PROGRAM P_Dialog
VAR
	nXPos 			: INT:=200; //pozycja popup na ekranie
	nYPos 			: INT:=200; //pozycja popup na ekranie
	fbOpenTrigger 	: R_TRIG;
	bClose 			: BOOL;
	fbCloseTrigger 	: R_TRIG;
	sMessage		: STRING;
	bOpen			: BOOL;
	sResult			: STRING;
	bVisible		: BOOl;
	tof1			: TOF;
	ftResult		: F_TRIG;
	bSwitchParameter: BOOL;
	nCount			: INT;
END_VAR

IF bSwitchParameter THEN
	sMessage:='Parameter text 111111';
ELSE
	sMessage:='Parameter text 222222';
END_IF


fbOpenTrigger(CLK :=bOpen);
IF fbOpenTrigger.Q THEN
	OpenMessageDialog(sMessage := sMessage);
	bOpen:=FALSE;
END_IF

fbCloseTrigger(CLK := bClose);
IF fbCloseTrigger.Q THEN
	nCount := nCount + 1;
	CloseMessageDialog();
	bClose:=FALSE;
END_IF


IF GVL.iMessageDialog <> 0 THEN
	GVL.result := GVL.iMessageDialog.GetResult();
END_IF


IF GVL.result = VisuElemsWinControls.Visu_DialogResult.OK THEN
	sResult:='You clicked OK'; 
END_IF

IF GVL.result = VisuElemsWinControls.Visu_DialogResult.Cancel THEN
	sResult:='You clicked Cancel'; 
END_IF

tof1(IN:=bVisible, PT:=T#1S);

bVisible:=FALSE;

END_PROGRAM

(* stored: Version 1.1.0.1, ProductVersion 3.1.4024.12
   POU P_Dialog: Id {b597f539-929f-4c55-92bb-bf76bd788e9c}, SpecialFunc None *)
